FUNCTION_BLOCK MachineSequenceStop EXTENDS MachineSequence IMPLEMENTS ZCore.ISequence
VAR
  _step : ZCore.Step(MachineStep.StopBegin, MachineStep.StopEnd);
  _timerSim : ZAux.Timer;
END_VAR

IF OnStart(_step) THEN
  ; // init custom sequence variables here ...
END_IF

REPEAT
  LogStep();

  CASE _step.Index OF
    (* -------------------------------------------------------------------------------------------------------------------------------- *)
    MachineStep.StopBegin:
    (* -------------------------------------------------------------------------------------------------------------------------------- *)
      IF _step.OnEntry()
      THEN
        _axis.ToolX.StopAsync(THIS^);
        _axis.TransportX.StopAsync(THIS^);  
			END_IF
      
      Await2(obj1:=_axis.ToolX, obj2:=_axis.TransportX, nextStep:=MachineStep.StopEnd);

    (* -------------------------------------------------------------------------------------------------------------------------------- *)
    MachineStep.StopEnd:
    (* -------------------------------------------------------------------------------------------------------------------------------- *)    
      SetBusy(FALSE);
  
  ELSE
    Abort('sequence contains unhandled step');
  END_CASE
UNTIL _step.IsNotRepeatable() OR_ELSE NOT Busy END_REPEAT

END_FUNCTION_BLOCK

(* stored: Version 1.1.0.1
   POU MachineSequenceStop: Id {3ca78a98-2874-404d-876f-3b0991d3ab4a}, SpecialFunc None *)
